// HOME mode chain (Core §6.2/§6.8 ST skeleton on FB_SequenceBase): establish the
// shared load-safe position, then complete. Finite (does not loop).
FUNCTION_BLOCK FB_PressDemoHome EXTENDS FB_SequenceBase
VAR
    {attribute 'OPC.UA.DA' := '0'}
    _outCmd : REFERENCE TO ST_PneumaticPressOutCmd;
    {attribute 'OPC.UA.DA' := '0'}
    _loadPosition : FB_PressDemoLoadPosition;
    _loadPositionRunning : BOOL;
END_VAR

METHOD M_Reset
M_ResetBase();
_loadPositionRunning := FALSE;
_loadPosition.M_Reset(BaseStepNo := 0);
END_METHOD

METHOD M_Run
IF NOT _attached THEN
    RETURN;
END_IF
CASE _step OF
    0:  // initialize
        M_Step(StepNo := 0, StepName := 'project.step.pressHomeInitialize',
            Awaits := 0, AwaitingLabel := '', TimeClass := E_TimeClass.WORK, ExpectedTime := T#0S);
        _outCmd.Homed := FALSE;
        _outCmd.ChangeoverCompleted := FALSE;
        _loadPositionRunning := FALSE;
        _retVal := E_StepResult.ADVANCE;
        M_Advance(OnAdvance := 900);
    900:  // shared load-safe position (composite step, §6.7)
        IF NOT _loadPositionRunning THEN
            _loadPosition.M_Reset(BaseStepNo := 900);
            _loadPositionRunning := TRUE;
        END_IF
        _loadPosition.M_Run();
        IF _loadPosition.Done THEN
            _loadPositionRunning := FALSE;
            _retVal := E_StepResult.ADVANCE;
        END_IF
        M_Advance(OnAdvance := 999);
    999:  // complete
        M_Step(StepNo := 999, StepName := 'project.step.pressHomeComplete',
            Awaits := 0, AwaitingLabel := '', TimeClass := E_TimeClass.WORK, ExpectedTime := T#0S);
        _outCmd.Homed := TRUE;
        M_Complete();
ELSE
    M_Fault(Reason := E_Reason.STEP_STALLED, DescriptionKey := 'std.error.undefinedStep');
END_CASE
END_METHOD

METHOD Setup : BOOL
VAR_INPUT
    Host : I_SequenceHost;
END_VAR
VAR_IN_OUT
    PressRam : FB_CylinderCM;
    Door : FB_CylinderCM;
    PartSlide : FB_CylinderCM;
    OutCmd : ST_PneumaticPressOutCmd;
END_VAR
_outCmd REF= OutCmd;
Setup := M_Attach(Host := Host) AND __ISVALIDREF(_outCmd)
    AND _loadPosition.Setup(Host := Host, PressRam := PressRam, Door := Door, PartSlide := PartSlide);
END_METHOD

END_FUNCTION_BLOCK

(* stored: Version 1.1.0.1
   POU FB_PressDemoHome: Id {27be7602-c702-dcca-822f-fb9fc2c72001}, SpecialFunc None
   Method M_Reset: Id {27be7602-c702-dcca-822f-fb9fc2c72003}
   Method M_Run: Id {27be7602-c702-dcca-822f-fb9fc2c72004}
   Method Setup: Id {27be7602-c702-dcca-822f-fb9fc2c72002} *)
